Universal Robots PolyScope program: fuerza.urp

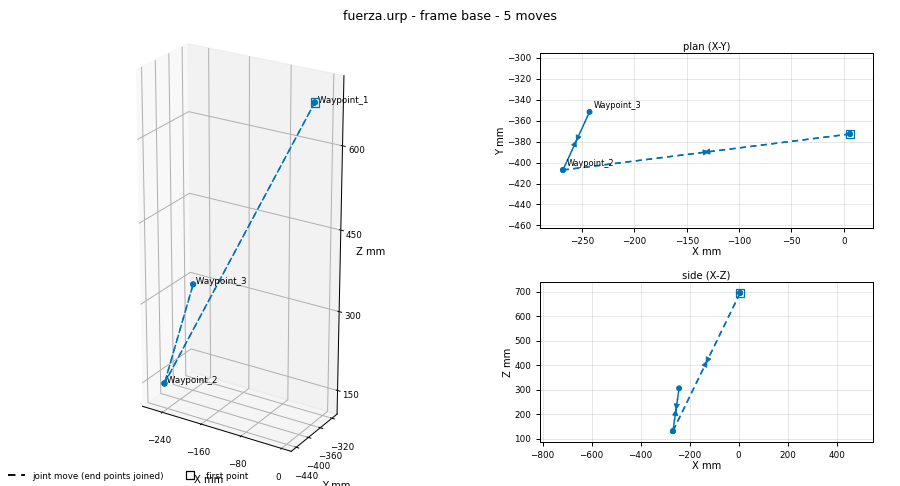
[picture p0: tool path of fuerza.urp in frame base, 5 of 5 moves have a stored position in this frame; points joined in program order, loops and branches not executed]
Program fuerza (installation=default directory=/programs createdIn=5.14.5 lastSavedIn=5.14.5 robotSerialNumber=20195300809)
Calibrated DH parameters: a=[-0.000085, -0.20076, -0.212369, 0.000121, -0.000118, 0]; d=[0.15185, -26.306375, 24.753047, 1.684739, 0.085386, 0.092088]; alpha=[1.572149, -0.00522, -0.011864, 1.571339, -1.571085, 0]; deltaTheta=[0, 0.599885, -0.513355, -0.086555, 0.000006, 0]
InitVariablesNode
BeforeStart
  URCap Gripper Activate (Robotiq_Grippers, Robotiq Inc.) dataModel(ResetAndActivateKey=false)
  URCap Gripper (Robotiq_Grippers, Robotiq Inc.) dataModel(position=0.0, force=0.0, speed=100.0, positionInDouble=0.0, forceInDouble=0.0, speedInDouble=100.0, slaveIds=[3], blocking=true)
  var_1 := 0
Robot Program (runOnlyOnce=true)
  MoveJ speed 60 deg/s, acceleration 80 deg/s^2 (useActiveTCP=true) feature=Base
    Waypoint Waypoint_1: TCP in base x=5.947 y=-372.7 z=694.671 mm, rx=-0.0179 ry=2.2101 rz=-2.2165 rad; joints [0.002, -89.999, 0, -90.001, 0.001, 0] deg; TCP offset x=0 y=0 z=150 mm, rx=0 ry=0 rz=0 rad
  MoveJ speed 60 deg/s, acceleration 80 deg/s^2 (useActiveTCP=true) feature=Base
    Waypoint Waypoint_2: TCP in base x=-268.281 y=-407.083 z=130.726 mm, rx=0.0255 ry=3.0678 rz=-0.0563 rad; joints [38.759, -41.295, 24.797, -71.606, -86.6, -50.187] deg
  URCap Gripper (Robotiq_Grippers, Robotiq Inc.) dataModel(position=100.0, force=100.0, speed=100.0, positionInDouble=100.0, forceInDouble=100.0, speedInDouble=100.0, slaveIds=[3], blocking=true)
  Script: socket_open("10.5.20.90",30003)
  var_1 := 1
  MoveJ speed 60 deg/s, acceleration 80 deg/s^2 (useActiveTCP=true) feature=Base
    Waypoint Waypoint_3: TCP in base x=-242.896 y=-351.576 z=305.767 mm, rx=-0.0971 ry=-3.0206 rz=0.3123 rad; joints [33.768, -54.333, 0.004, -47.462, -84.671, -51.478] deg
    var_1 := 0
  MoveJ speed 60 deg/s, acceleration 80 deg/s^2 (useActiveTCP=true) feature=Base
    Waypoint Waypoint_2: TCP in base x=-268.281 y=-407.083 z=130.726 mm, rx=0.0255 ry=3.0678 rz=-0.0563 rad; joints [38.759, -41.295, 24.797, -71.606, -86.6, -50.187] deg
    URCap Gripper (Robotiq_Grippers, Robotiq Inc.) dataModel(position=0.0, force=0.0, speed=100.0, positionInDouble=0.0, forceInDouble=0.0, speedInDouble=100.0, slaveIds=[3], blocking=true)
  MoveJ speed 60 deg/s, acceleration 80 deg/s^2 (useActiveTCP=true) feature=Base
    Waypoint Waypoint_1: TCP in base x=5.947 y=-372.7 z=694.671 mm, rx=-0.0179 ry=2.2101 rz=-2.2165 rad; joints [0.002, -89.999, 0, -90.001, 0.001, 0] deg
Thread Thread_1 (runOnlyOnce=false)
  Loop While (checkContinuously=false) expression=var_1≟1
    f := force()
    ff := to_str(f)
    Script: socket_send_line(ff)
    Wait Sleep waitTime=0.01
